{attribute addProperty BoxType "EPP2038-0001-0016"}
{attribute addProperty Id "Diag_ChannelAT %I*ARRAY[0..7] OF Diag_Channel_E4AEF59E6480ChannelAT %Q*ARRAY[0..7] OF Channel_7F374EB06480WcStateAT %I*WcState_F855686C1620InfoDataAT %I*InfoData_192954DE1620"}
{attribute addProperty CRC "3530358484"}
{attribute addProperty SizeInBites "160"}
{attribute addProperty SizeInBytes "20"}
TYPE EPP2038_309488D0 :
STRUCT
	{attribute addProperty Name "Diag_Channel"}
	Diag_Channel : ARRAY[0..7] OF Diag_Channel_E4AEF59E;
	{attribute addProperty Name "Channel"}
	Channel : ARRAY[0..7] OF Channel_7F374EB0;
	{attribute addProperty Name "WcState"}
	WcState : WcState_F855686C;
	{attribute addProperty Name "InfoData"}
	InfoData : InfoData_192954DE;
END_STRUCT
END_TYPE

(* stored: Version 1.2.0.0, ProductVersion 3.1.4024.9
   DUT EPP2038_309488D0: Id {8ce360a4-6545-4cdf-af2e-15201dd77ef4} *)
